FUNCTION_BLOCK IOs
VAR_INPUT
	//850KF3
	x_EB_KO1: BOOL;
	x_Reset_KO1: BOOL;
	x_EB_KO2: BOOL;
	x_Reset_KO2: BOOL;
	x_EB_VD_PU: BOOL;
	x_EB_KD_PU: BOOL;
	x_EB_GW_PU: BOOL;
	x_EB_Abtauen_PU: BOOL;
	x_EB_KWP_PU: BOOL;
	x_EB_RW_PU: BOOL;
	x_EB_Speichernachheizung: BOOL;
	x_EB_KWP_PU2: BOOL;
	x_EB_KWP_PU3: BOOL;
	x_EB_TWW_PU: BOOL;
	x_EB_Zirk_PU: BOOL;
	x_EB_HG1_PU: BOOL;
	//850KF6
	f_RS_VD_PU: REAL;
	f_RS_KD_PU: REAL;
	f_RS_Hochhaltung: REAL;
	f_RS_Tiefhaltung: REAL;
	f_RS_TWW_PU: REAL;
	f_RS_RW: REAL;
	f_RS_MV_RW: REAL;
	f_RS_Vorlauf_Kuehlen: REAL;
	//850KF6.1
	x_EEV_EN: BOOL;
	f_RS_EEV: REAL;
	x_EEV_Kalibrieren: BOOL;
	x_EEV_SW_Reset: BOOL;
	//851KF2
	x_EB_HG2_PU: BOOL;
	x_EB_HG3_PU: BOOL;
	x_EB_HG4_PU: BOOL;
	x_EB_Spindelheizung: BOOL;
	x_EB_RW: BOOL;
	x_EB_AV_TWW_HWP: BOOL;
	x_EB_AV_RW: BOOL;
	x_EB_AV_RW_Primaer: BOOL;
	x_EB_AV_VL_HWP: BOOL;
	x_EB_AV_Abtauung: BOOL;
	x_EB_AV_Primaerkreis: BOOL;
	x_EB_AV_Kuehlung: BOOL;
	x_EB_AV_Kuehlung2: BOOL;
	x_EB_AV_RL_HWP: BOOL;
	x_EB_AV_RW_Rueckkuehler: BOOL;
	x_EB_AV_TWW: BOOL;
	//851KF2.1
	x_EB_AV_TWW_Notheizung: BOOL;
	x_EB_AV_RL_TWW: BOOL;
	x_EB_UV_HG1: BOOL;
	x_EB_UV_HG2: BOOL;
	x_EB_UV_HG3: BOOL;
	x_EB_UV_HG4: BOOL;
	x_EB_ZH: BOOL;
	x_EB_HWP_NH: BOOL;
	x_EB_TWW_NH: BOOL;
	x_EB_Oelsumpfheizung: BOOL;
	//851KF4.1
	f_RS_MV_HG1: REAL;
	f_RS_MV_HG2: REAL;
	f_RS_MV_HG3: REAL;
	f_RS_MV_HG4: REAL;
	f_RS_MV_ZH: REAL;
	f_RS_ZH: REAL;
	f_RS_EEV_Siemens: REAL;
END_VAR
VAR_OUTPUT
	//850KF2
	x_BM_USV: BOOL;
	x_BM_KO1: BOOL;
	x_BM_SHD_KO1: BOOL;
	x_BM_WS_KO1: BOOL;
	x_BM_KO2: BOOL;
	x_BM_SHD_KO2: BOOL;
	x_BM_WS_KO2: BOOL;
	x_BM_VD_PU_Betrieb: BOOL;
	x_BM_KD_PU_Betrieb: BOOL;
	x_BM_P_Primaer: BOOL;
	x_BM_STW_Primaer: BOOL;
	x_BM_EVU: BOOL;
	x_BM_FG_HWP: BOOL;
	x_BM_GW_PU_Betrieb: BOOL;
	x_BM_Abtauen_PU_Betrieb: BOOL;
	x_BM_KWP_PU_Betrieb: BOOL;
	//850KF4
	f_MT_HG1: REAL;
	f_MT_HG2: REAL;
	f_MT_SG: REAL;
	f_MT_VD_Ein: REAL;
	f_MT_VD_Aus: REAL;
	f_MT_KD_Ein: REAL;
	f_MT_KD_Aus: REAL;
	f_MT_FG: REAL;
	//850KF4.1
	f_MT_AT: REAL;
	f_MT_HWP_Oben: REAL;
	f_MT_HWP_Unten: REAL;
	f_MT_LuftEinRueckkuehler: REAL;
	f_MT_LuftAusRueckkuehler: REAL;
	f_MT_RW_Ein: REAL;
	f_MT_RW_Aus: REAL;
	f_MT_Gehaeuse: REAL;
	//850KF5
	f_MP_ND: REAL;
	f_MP_HD: REAL;
	f_RM_Kaeltemittelsensor: REAL;
	f_SW_HWP: REAL;
	f_SW_KWP: REAL;
	//851KF0
	x_BM_RW_PU_Betrieb: BOOL;
	x_BM_Speichernachheizung_Betrieb: BOOL;
	x_BM_KWP_PU_Betrieb2: BOOL;
	x_BM_KWP_PU_Betrieb3: BOOL;
	x_BM_TWW_PU_Betrieb: BOOL;
	x_BM_Zirk_PU_Betrieb: BOOL;
	x_BM_HG1_PU_Betrieb: BOOL;
	x_BM_HG2_PU_Betrieb: BOOL;
	x_BM_HG3_PU_Betrieb: BOOL;
	x_BM_HG4_PU_Betrieb: BOOL;
	x_BM_Frischwasser_Alarm: BOOL;
	x_BM_RW_Betrieb: BOOL;
	x_BM_RW_Alarm: BOOL;
	x_BM_STW_KWP: BOOL;
	x_BM_STW_RW: BOOL;
	x_BM_Tempwaechter_HG1: BOOL;
	//851KF1
	x_BM_Tempwaechter_HG2: BOOL;
	x_BM_Tempwaechter_HG3: BOOL;
	x_BM_Tempwaechter_HG4: BOOL;
	x_BM_Feuchteschalter_HG1: BOOL;
	x_BM_Feuchteschalter_HG2: BOOL;
	x_BM_Feuchteschalter_HG3: BOOL;
	x_BM_Feuchteschalter_HG4: BOOL;
	x_BM_FG_KWP: BOOL;
	x_BM_FG_TWW: BOOL;
	x_BM_ZH_Netrieb: BOOL;
	x_BM_ZH_Alarn: BOOL;
	//851KF3
	f_MT_RW_WT_Aus_Primaer: REAL;
	f_MT_RW_WT_Aus: REAL;
	f_MT_RW_RL: REAL;
	f_MT_VL_HG1: REAL;
	f_MT_VL_HG2: REAL;
	f_MT_VL_HG3: REAL;
	f_MT_VL_HG4: REAL;
	f_MT_TWW_Unten: REAL;
	//851KF4
	f_MT_TWW_Oben: REAL;
	f_MT_TWW_VL: REAL;
	f_MT_VL_Kuehlung: REAL;
	
	f_MT_KWP_Oben: REAL;
	f_MT_KWP_Unten: REAL;
	f_MT_VL_HG: REAL;
	//851KF6
	
	//851KF6.1
END_VAR
VAR
	DI_850KF2: DI_16;
	DO_850KF3: DO_16;
	AI_850KF4: AI_8_Temp;
	AI_850KF4_1: AI_8_Temp;
	AI_850KF5: AI_8_4_20mA;
	AO_850KF6: AO_8;
	SM_850KF6_1: EEV_Schrittmotor;
	DI_851KF0: DI_16;
	DI_851KF1: DI_16;
	DO_851KF2: DO_16;
	DO_851KF2_1: DO_16;
	AI_851KF3: AI_8_Temp;
	AI_851KF4: AI_8_Temp;
	AO_851KF4_1: AO_8;
	AI_851KF6: AI_8_Temp;
	EM_851KF6_1: Elektromessung;
END_VAR

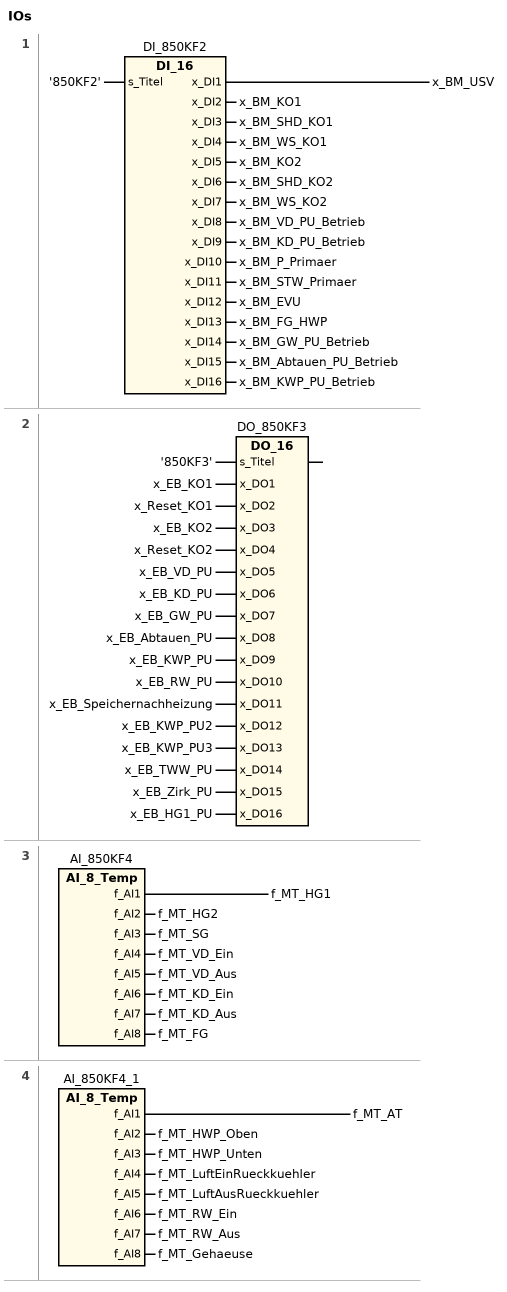
// NETWORK 1
DI_850KF2(
    s_Titel := '850KF2',
    x_DI2 => x_BM_KO1,
    x_DI3 => x_BM_SHD_KO1,
    x_DI4 => x_BM_WS_KO1,
    x_DI5 => x_BM_KO2,
    x_DI6 => x_BM_SHD_KO2,
    x_DI7 => x_BM_WS_KO2,
    x_DI8 => x_BM_VD_PU_Betrieb,
    x_DI9 => x_BM_KD_PU_Betrieb,
    x_DI10 => x_BM_P_Primaer,
    x_DI11 => x_BM_STW_Primaer,
    x_DI12 => x_BM_EVU,
    x_DI13 => x_BM_FG_HWP,
    x_DI14 => x_BM_GW_PU_Betrieb,
    x_DI15 => x_BM_Abtauen_PU_Betrieb,
    x_DI16 => x_BM_KWP_PU_Betrieb); // DI_16
x_BM_USV := DI_850KF2.x_DI1;

// NETWORK 2
DO_850KF3(
    s_Titel := '850KF3',
    x_DO1 := x_EB_KO1,
    x_DO2 := x_Reset_KO1,
    x_DO3 := x_EB_KO2,
    x_DO4 := x_Reset_KO2,
    x_DO5 := x_EB_VD_PU,
    x_DO6 := x_EB_KD_PU,
    x_DO7 := x_EB_GW_PU,
    x_DO8 := x_EB_Abtauen_PU,
    x_DO9 := x_EB_KWP_PU,
    x_DO10 := x_EB_RW_PU,
    x_DO11 := x_EB_Speichernachheizung,
    x_DO12 := x_EB_KWP_PU2,
    x_DO13 := x_EB_KWP_PU3,
    x_DO14 := x_EB_TWW_PU,
    x_DO15 := x_EB_Zirk_PU,
    x_DO16 := x_EB_HG1_PU); // DO_16

// NETWORK 3
AI_850KF4(
    f_AI2 => f_MT_HG2,
    f_AI3 => f_MT_SG,
    f_AI4 => f_MT_VD_Ein,
    f_AI5 => f_MT_VD_Aus,
    f_AI6 => f_MT_KD_Ein,
    f_AI7 => f_MT_KD_Aus,
    f_AI8 => f_MT_FG); // AI_8_Temp
f_MT_HG1 := AI_850KF4.f_AI1;

// NETWORK 4
AI_850KF4_1(
    f_AI2 => f_MT_HWP_Oben,
    f_AI3 => f_MT_HWP_Unten,
    f_AI4 => f_MT_LuftEinRueckkuehler,
    f_AI5 => f_MT_LuftAusRueckkuehler,
    f_AI6 => f_MT_RW_Ein,
    f_AI7 => f_MT_RW_Aus,
    f_AI8 => f_MT_Gehaeuse); // AI_8_Temp
f_MT_AT := AI_850KF4_1.f_AI1;

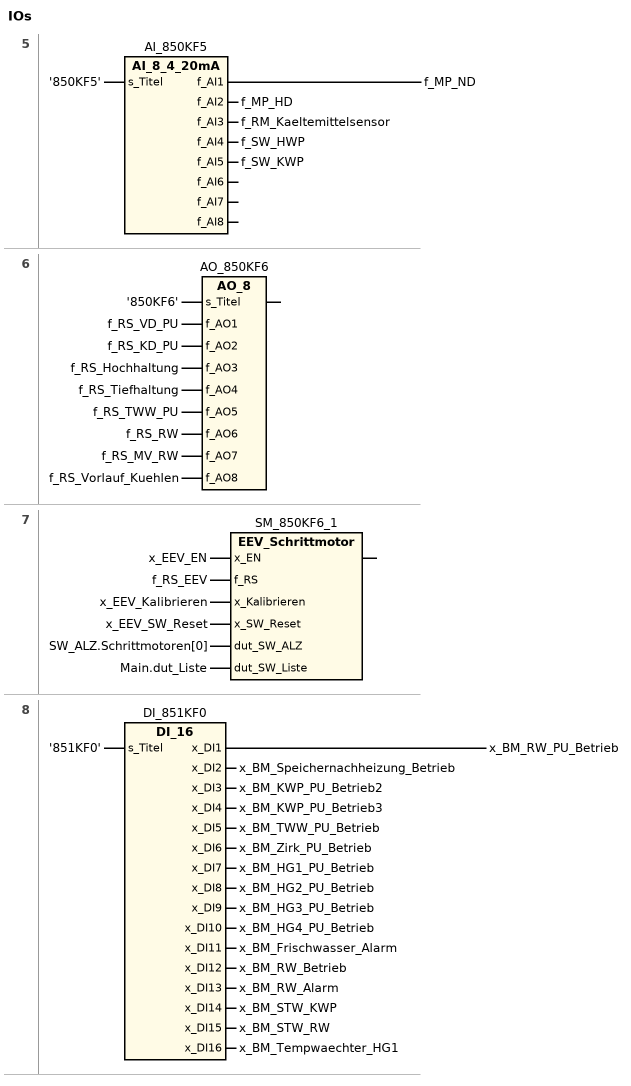
// NETWORK 5
AI_850KF5(
    s_Titel := '850KF5',
    f_AI2 => f_MP_HD,
    f_AI3 => f_RM_Kaeltemittelsensor,
    f_AI4 => f_SW_HWP,
    f_AI5 => f_SW_KWP); // AI_8_4_20mA
f_MP_ND := AI_850KF5.f_AI1;

// NETWORK 6
AO_850KF6(
    s_Titel := '850KF6',
    f_AO1 := f_RS_VD_PU,
    f_AO2 := f_RS_KD_PU,
    f_AO3 := f_RS_Hochhaltung,
    f_AO4 := f_RS_Tiefhaltung,
    f_AO5 := f_RS_TWW_PU,
    f_AO6 := f_RS_RW,
    f_AO7 := f_RS_MV_RW,
    f_AO8 := f_RS_Vorlauf_Kuehlen); // AO_8

// NETWORK 7
SM_850KF6_1(
    x_EN := x_EEV_EN,
    f_RS := f_RS_EEV,
    x_Kalibrieren := x_EEV_Kalibrieren,
    x_SW_Reset := x_EEV_SW_Reset,
    dut_SW_ALZ := SW_ALZ.Schrittmotoren[0],
    dut_SW_Liste := Main.dut_Liste); // EEV_Schrittmotor

// NETWORK 8
DI_851KF0(
    s_Titel := '851KF0',
    x_DI2 => x_BM_Speichernachheizung_Betrieb,
    x_DI3 => x_BM_KWP_PU_Betrieb2,
    x_DI4 => x_BM_KWP_PU_Betrieb3,
    x_DI5 => x_BM_TWW_PU_Betrieb,
    x_DI6 => x_BM_Zirk_PU_Betrieb,
    x_DI7 => x_BM_HG1_PU_Betrieb,
    x_DI8 => x_BM_HG2_PU_Betrieb,
    x_DI9 => x_BM_HG3_PU_Betrieb,
    x_DI10 => x_BM_HG4_PU_Betrieb,
    x_DI11 => x_BM_Frischwasser_Alarm,
    x_DI12 => x_BM_RW_Betrieb,
    x_DI13 => x_BM_RW_Alarm,
    x_DI14 => x_BM_STW_KWP,
    x_DI15 => x_BM_STW_RW,
    x_DI16 => x_BM_Tempwaechter_HG1); // DI_16
x_BM_RW_PU_Betrieb := DI_851KF0.x_DI1;

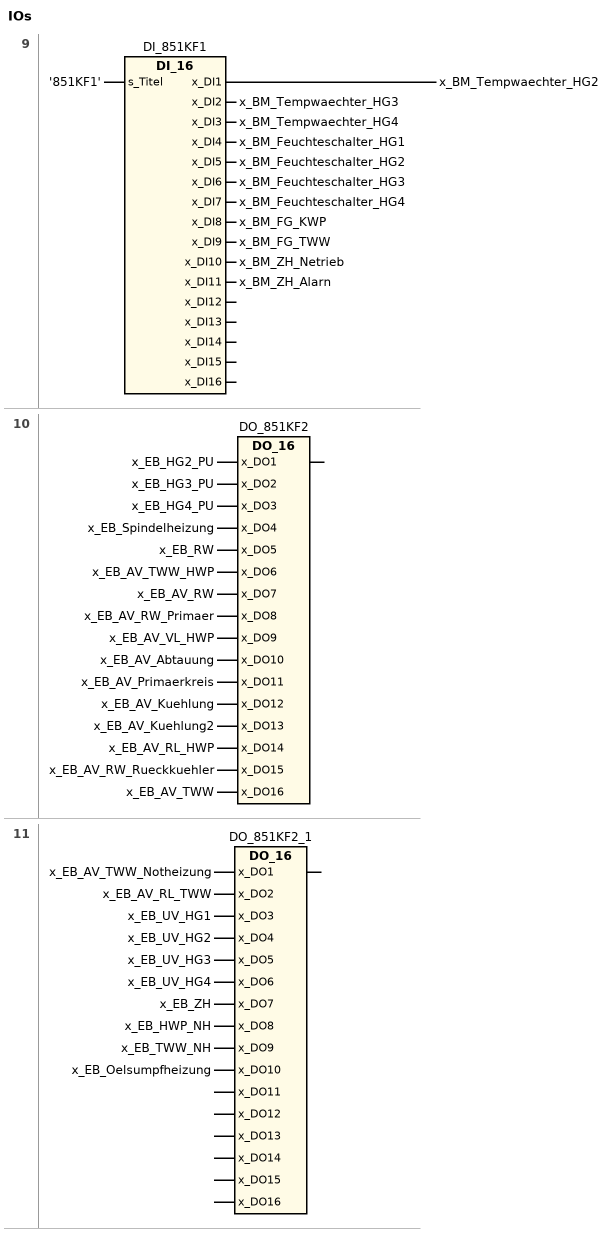
// NETWORK 9
DI_851KF1(
    s_Titel := '851KF1',
    x_DI2 => x_BM_Tempwaechter_HG3,
    x_DI3 => x_BM_Tempwaechter_HG4,
    x_DI4 => x_BM_Feuchteschalter_HG1,
    x_DI5 => x_BM_Feuchteschalter_HG2,
    x_DI6 => x_BM_Feuchteschalter_HG3,
    x_DI7 => x_BM_Feuchteschalter_HG4,
    x_DI8 => x_BM_FG_KWP,
    x_DI9 => x_BM_FG_TWW,
    x_DI10 => x_BM_ZH_Netrieb,
    x_DI11 => x_BM_ZH_Alarn); // DI_16
x_BM_Tempwaechter_HG2 := DI_851KF1.x_DI1;

// NETWORK 10
DO_851KF2(
    x_DO1 := x_EB_HG2_PU,
    x_DO2 := x_EB_HG3_PU,
    x_DO3 := x_EB_HG4_PU,
    x_DO4 := x_EB_Spindelheizung,
    x_DO5 := x_EB_RW,
    x_DO6 := x_EB_AV_TWW_HWP,
    x_DO7 := x_EB_AV_RW,
    x_DO8 := x_EB_AV_RW_Primaer,
    x_DO9 := x_EB_AV_VL_HWP,
    x_DO10 := x_EB_AV_Abtauung,
    x_DO11 := x_EB_AV_Primaerkreis,
    x_DO12 := x_EB_AV_Kuehlung,
    x_DO13 := x_EB_AV_Kuehlung2,
    x_DO14 := x_EB_AV_RL_HWP,
    x_DO15 := x_EB_AV_RW_Rueckkuehler,
    x_DO16 := x_EB_AV_TWW); // DO_16

// NETWORK 11
DO_851KF2_1(
    x_DO1 := x_EB_AV_TWW_Notheizung,
    x_DO2 := x_EB_AV_RL_TWW,
    x_DO3 := x_EB_UV_HG1,
    x_DO4 := x_EB_UV_HG2,
    x_DO5 := x_EB_UV_HG3,
    x_DO6 := x_EB_UV_HG4,
    x_DO7 := x_EB_ZH,
    x_DO8 := x_EB_HWP_NH,
    x_DO9 := x_EB_TWW_NH,
    x_DO10 := x_EB_Oelsumpfheizung); // DO_16

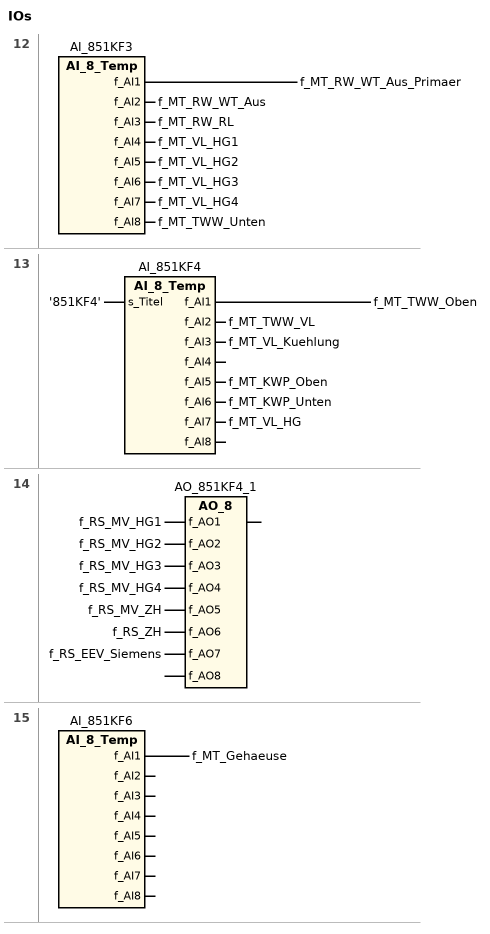
// NETWORK 12
AI_851KF3(
    f_AI2 => f_MT_RW_WT_Aus,
    f_AI3 => f_MT_RW_RL,
    f_AI4 => f_MT_VL_HG1,
    f_AI5 => f_MT_VL_HG2,
    f_AI6 => f_MT_VL_HG3,
    f_AI7 => f_MT_VL_HG4,
    f_AI8 => f_MT_TWW_Unten); // AI_8_Temp
f_MT_RW_WT_Aus_Primaer := AI_851KF3.f_AI1;

// NETWORK 13
AI_851KF4(
    s_Titel := '851KF4',
    f_AI2 => f_MT_TWW_VL,
    f_AI3 => f_MT_VL_Kuehlung,
    f_AI5 => f_MT_KWP_Oben,
    f_AI6 => f_MT_KWP_Unten,
    f_AI7 => f_MT_VL_HG); // AI_8_Temp
f_MT_TWW_Oben := AI_851KF4.f_AI1;

// NETWORK 14
AO_851KF4_1(
    f_AO1 := f_RS_MV_HG1,
    f_AO2 := f_RS_MV_HG2,
    f_AO3 := f_RS_MV_HG3,
    f_AO4 := f_RS_MV_HG4,
    f_AO5 := f_RS_MV_ZH,
    f_AO6 := f_RS_ZH,
    f_AO7 := f_RS_EEV_Siemens); // AO_8

// NETWORK 15
AI_851KF6(); // AI_8_Temp
f_MT_Gehaeuse := AI_851KF6.f_AI1;

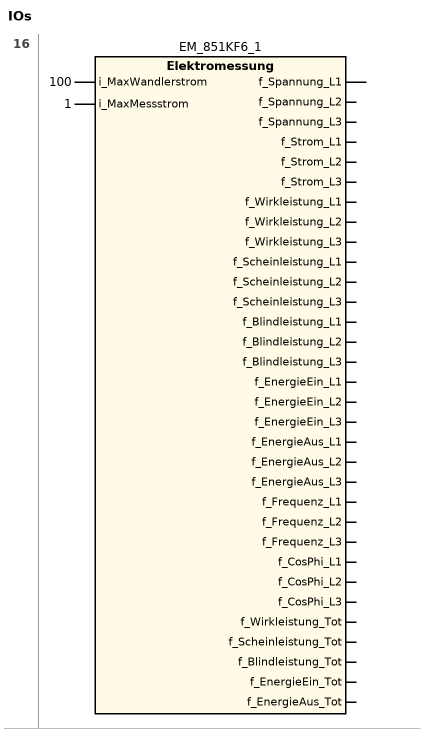
// NETWORK 16
EM_851KF6_1(i_MaxWandlerstrom := 100, i_MaxMessstrom := 1); // Elektromessung

END_FUNCTION_BLOCK

(* stored: Version 1.1.0.1, ProductVersion 3.1.4022.6
   POU IOs: Id {2593276f-7c06-4336-baea-3e909951fac0}, SpecialFunc None *)
